IF NOT UseEnableWire THEN
	IF checkInitMultiplex() THEN
		RETURN;
	END_IF
ELSE
	IF NOT enableInstanceSet THEN
		RETURN;
	END_IF
END_IF
CASE _iState OF

RUN_DEVICE:
	//check if time are over
	IF TimeToRead < TICKS.GetTick(xDummy:= TRUE) AND haveToRead THEN 
		readRequest.request := TRUE;
		haveToRead := FALSE;
		TimeToReadOver := TRUE;
	END_IF
	IF UseEnableWire THEN
		IF NOT TimeToReadOver THEN
			RETURN;
		END_IF
	ELSE
		IF NOT checkReadTimeMultiplex(ADR(readRequest)) OR NOT TimeToReadOver THEN
			RETURN;
		END_IF
	END_IF
	ReadTime := TICKS.GetTick(xDummy:= TRUE);
	TimeToReadOver := FALSE;
	waitForDone := FALSE;
	IF NOT (setWire() = SET_SLAVE_NUM_RETURN.NUM_IO) AND UseEnableWire  THEN
		RETURN;
	END_IF
	//time over and on the bus... now read
	//read RH
	IF checkRead(pbyBuffer:= ADR(buffer), nBufferLen:= 3(*SIZEOF(buffer)*)) = ERROR_RET_VAL THEN
		ReadHuminityErrorRate := ReadHuminityErrorRate + 1;
		RETURN; 
	END_IF
	buffercrc[1] := buffer[0];
	buffercrc[2] := buffer[1];
	buffercrc[3] := buffer[2];
	buffercrc[0] := 0;
	crc := OSCAT_BASIC.CRC_GEN(
	PT:= ADR(buffercrc), 
	SIZE:= TO_INT(SIZEOF(buffercrc)), 
	PL:= 8, 
	PN:= 16#31, 
	INIT:= 0, 
	REV_IN:= FALSE, 
	REV_OUT:= FALSE, 
	XOR_OUT:= 0);
	IF crc = 0 THEN
		//checkRead(pbyBuffer:= ADR(buffer), nBufferLen:= SIZEOF(buffer));
		myData.Humidity := (((DWORD_TO_LREAL(OSCAT_BASIC.DWORD_OF_BYTE(B3:= 0, B2:= 0, B1:= buffer[0], B0:= buffer[1]))*125)/65536))-6;
		//read temp with command
		buffer[0] := COMMAND_READ_TEMP_FROM_PREVIOUS_RH;
		IF checkWrite(pbyBuffer:= ADR(buffer), nBufferLen:= 1) = ERROR_RET_VAL THEN //write just one command
			WriteTempReadErrorRate := WriteTempReadErrorRate + 1;
			RETURN; 
		END_IF
		IF checkRead(pbyBuffer:= ADR(buffer), nBufferLen:=2 (* SIZEOF(buffer)*)) = ERROR_RET_VAL THEN 
			ReadTempErrorRate := ReadTempErrorRate + 1;
		RETURN;
		END_IF
		myData.Temperatur := ((DWORD_TO_LREAL(OSCAT_BASIC.DWORD_OF_BYTE(B3:= 0, B2:= 0, B1:= buffer[0], B0:= buffer[1]))*175.72)/65536)-46.85;
		
		myData.absHumidity  := OSCAT_BUILDING.DEW_CON(RH:=LREAL_TO_REAL(myData.Humidity) , T:=LREAL_TO_REAL(myData.Temperatur) );
		myData.dewPoint := OSCAT_BUILDING.DEW_TEMP(RH:= LREAL_TO_REAL(myData.Humidity), T:=LREAL_TO_REAL(myData.Temperatur ));
	ELSE
		CRCErrorRate := CRCErrorRate + 1;
		goError(ReadWrite:=FALSE);
	END_IF
	releaseWire();

END_CASE
END_METHOD

METHOD BeforeWriteOutputs : INT
VAR

buffer:ARRAY[0..1]OF BYTE;

SystemTime: CAA.TICK;

END_VAR
SUPER^.BeforeWriteOutputs();

IF NOT UseEnableWire THEN
	IF checkInitMultiplex() THEN
		RETURN;
	END_IF
ELSE
	IF NOT enableInstanceSet THEN
		RETURN;
	END_IF
END_IF

CASE _iState OF
START_DEVICE:
	//check if time is over
	//writeRequest.request := requestOnInit;
	waitForDone := FALSE;
	writeRequest.request := TRUE;
	IF checkWriteTimeMultiplex(ADR(writeRequest)) = FALSE AND NOT UseEnableWire THEN
		RETURN;// i am not on the bus
	END_IF
	buffer[0] := COMMAND_WRITE_RESISTER_1;
	buffer[1] := controlRegister; 
	
	IF NOT (setWire() = SET_SLAVE_NUM_RETURN.NUM_IO) AND UseEnableWire THEN
		RETURN;
	END_IF
	checkWrite(pbyBuffer:= ADR(buffer), nBufferLen:= SIZEOF(buffer));
	IF _iState<>ERROR_DEVICE THEN
		_iState := RUN_DEVICE;
		//requestOnInit := FALSE;//init successful	
	END_IF
	releaseWire();		
RUN_DEVICE:
	SystemTime := TICKS.GetTick(xDummy:= TRUE);
	IF NextMeasuerment < SystemTime AND NOT waitForDone THEN 
		NextMeasuerment := timeMeasurment + SystemTime;
		waitForDone := TRUE; 
		writeRequest.request := TRUE;
		WriteRequestHuminity := TRUE;
	END_IF
	IF UseEnableWire THEN
		IF NOT WriteRequestHuminity THEN
			RETURN;
		END_IF
	ELSE
		IF NOT checkReadTimeMultiplex(ADR(writeRequest)) OR NOT WriteRequestHuminity THEN
			RETURN;
		END_IF
	END_IF
	WriteRequestHuminity := FALSE;
	//new time for Read the conversation
	TimeToRead := timePreset + TICKS.GetTick(xDummy:= TRUE);
	haveToRead := TRUE;

	IF NOT (setWire() = SET_SLAVE_NUM_RETURN.NUM_IO) AND UseEnableWire THEN
		RETURN;
	END_IF
	
	buffer[0] := COMMAND_MEASURE_RH_NO_HOLD_MASTER;
	IF checkWrite(pbyBuffer:= ADR(buffer), nBufferLen:= 1) = ERROR_RET_VAL THEN //write just one byte!
		WriteTempReadErrorRate := WriteTempReadErrorRate + 1;
	END_IF
	WriteTime := TICKS.GetTick(xDummy:= TRUE);
	releaseWire();
END_CASE
END_METHOD

METHOD Initialize : UDINT
VAR_INPUT
	wModuleType : UINT;
	dwInstance : UDINT;
	pConnector : POINTER TO IoConfigConnector;
END_VAR
VAR
	pParam: POINTER TO IoConfigParameter;		
	udiResult: UDINT;
	config:USINT;
END_VAR
SUPER^.Initialize(wModuleType, dwInstance, pConnector);
usiAddress := 16#40;
//get config
pParam := ConfigGetParameter(_pConnector, 20);



config:= IoStandard.ConfigGetParameterValueByte(pParam, ADR(udiResult));
CASE config OF//see Datasheet Page 26 for config
	//control Register --> resoulution
	0:	controlRegister := 2#1;
		timePreset := 8;//ms
	1:	controlRegister := 2#10000000;
		timePreset := 12;//ms
	2:	controlRegister := 2#10000001;
		timePreset := 12;//ms
	3:	controlRegister := 2#0;
		timePreset := 25;//ms
END_CASE

//time between Measurments
pParam := ConfigGetParameter(_pConnector, 21);
timeMeasurment := IoStandard.ConfigGetParameterValueDWord(pParam, ADR(udiResult));
//disable auto read
readRequest.timePreset := 16#FFFFFFFF; 
 
stateAfterError := START_DEVICE;
stateAfterInit := START_DEVICE;
END_METHOD

END_FUNCTION_BLOCK

// Function Blocks/BMP280
FUNCTION_BLOCK BMP280 EXTENDS I2C_BASE
VAR_INPUT

END_VAR
VAR_OUTPUT
	myData:BMP280Data;
	configWrong: BOOL;
END_VAR
VAR


	dig_T1: LREAL;
    dig_T2: LREAL;
    dig_T3: LREAL;
	 
    dig_P1: LREAL;
    dig_P2: LREAL;
    dig_P3: LREAL;
    dig_P4: LREAL;
    dig_P5: LREAL;
    dig_P6: LREAL;
    dig_P7: LREAL;
    dig_P8: LREAL;
    dig_P9: LREAL;

	t_fine:DINT;
	
	tempOversampling: USINT;
	pressureOversampling: USINT;

	iirFilter:USINT;
	standbyTime:USINT;
	controlRegister:BYTE;
	writeControlRegister:BOOL;
	operationMode:BYTE;
	//diffrenz for read the next value in ms
	nextForcedDiff:UDINT;
	//next time to write forced
	nextForced: CAA.TICK;
	//wrong device!
	wrongDevice: BOOL;


END_VAR
VAR_TEMP	
END_VAR

VAR CONSTANT 
	
BMP280_REGISTER_DIG_T1:USINT := 16#88;
BMP280_REGISTER_DIG_T2:USINT := 16#8A;
BMP280_REGISTER_DIG_T3:USINT := 16#8C;

BMP280_REGISTER_DIG_P1:USINT := 16#8E;
BMP280_REGISTER_DIG_P2:USINT := 16#90;
BMP280_REGISTER_DIG_P3:USINT := 16#92;
BMP280_REGISTER_DIG_P4:USINT := 16#94;
BMP280_REGISTER_DIG_P5:USINT := 16#96;
BMP280_REGISTER_DIG_P6:USINT := 16#98;
BMP280_REGISTER_DIG_P7:USINT := 16#9A;
BMP280_REGISTER_DIG_P8:USINT := 16#9C;
BMP280_REGISTER_DIG_P9:USINT := 16#9E;



BMP280_REGISTER_CHIPID:USINT := 16#D0;
BMP280_REGISTER_VERSION :USINT := 16#D1;
BMP280_REGISTER_SOFTRESET :USINT := 16#E0;


BMP280_REGISTER_CONTROL :USINT := 16#F4;
BMP280_REGISTER_CONFIG :USINT := 16#F5;
BMP280_REGISTER_PRESSURE_DATA :USINT := 16#F7;
BMP280_REGISTER_TEMP_DATA :USINT := 16#FA;

BMP_280_DEVICE_ID:USINT:=16#58;

TEMP_OVERSAMPLING_MAX:USINT:=5;
PRESSURE_OVERSAMPLING_MAX:USINT:=5;

IIR_FILTER_MAX:USINT:=4;
STANDBY_TIME_MAX:USINT:=7;
BMP280_NORMAL_MODE:USINT:=2#11;
BMP280_FORCED_MODE:USINT:=2#01;
BMP280_SLEEP_MODE:USINT:=2#00;

TEMPERATURE_OFF:UDINT:=16#80000;
PRESSURE_OFF:UDINT:=16#80000;




END_VAR

SUPER^();

CASE _iState OF
	RUN_DEVICE:
		IF operationMode = BMP280_FORCED_MODE THEN
			IF nextForced < TICKS.GetTick(xDummy:= TRUE) THEN
				//set next read
				nextForced := nextForcedDiff + TICKS.GetTick(xDummy:= TRUE);
				setForcedMode();
				
			END_IF 
		ELSE
			nextForced := nextForcedDiff + TICKS.GetTick(xDummy:= TRUE);
		END_IF
END_CASE

METHOD AfterReadInputs : INT
VAR
	sensorData: ARRAY[0..7] OF BYTE;	
	rawTempSensor:UDINT;
	rawTemp:LREAL;
	rawPressureSensor:UDINT;
	rawPressure:LREAL;
	rawHumiditySensor:UDINT;
	rawHumidity:LREAL;
	var1, var2, p, var_H:LREAL;
	tError, hError, pError: BOOL;
	//dd:LREAL;
END_VAR
SUPER^.AfterReadInputs();

IF checkInitMultiplex() THEN
	RETURN;
END_IF
CASE _iState OF
START_INIT:
	readRequest.request := TRUE;
	
	//check if time are over
	IF NOT checkReadTimeMultiplex(ADR(readRequest)) THEN
		RETURN;
	END_IF
	initCalibration();

	IF _iState<>ERROR_DEVICE THEN
		_iState := START_DEVICE;

	END_IF
RUN_DEVICE:
	//check if time are over
	IF NOT checkReadTimeMultiplex(ADR(readRequest)) THEN
		RETURN;
	END_IF
	(*read all sensor Data*)
	IF checkReadRegister(BMP280_REGISTER_PRESSURE_DATA, ADR(sensorData),6) < 0 THEN
		RETURN;
	END_IF
	
	rawTempSensor:=0;
	rawTempSensor:=SHL(BYTE_TO_UDINT(sensorData[3]),16);
	rawTempSensor:=rawTempSensor OR SHL(BYTE_TO_UDINT(sensorData[4]),8);
	rawTempSensor:=rawTempSensor OR BYTE_TO_UDINT(sensorData[5]);
	rawTempSensor:= SHR(rawTempSensor,4);
	//if Sensor value off and sensor switched on(no power)
	IF rawTempSensor = TEMPERATURE_OFF AND tempOversampling >0 THEN
		goError(ReadWrite := TRUE);
		RETURN;
	END_IF
	IF rawTempSensor <> 16#80000 THEN
		rawTemp:=UDINT_TO_REAL(rawTempSensor);
		var1  := (rawTemp/16384.0 - dig_T1/1024.0) * dig_T2;
		var2  := ((rawTemp/131072.0 - dig_T1/8192.0) *   (rawTemp/131072.0 -  dig_T1/8192.0)) * dig_T3;
		t_fine := LREAL_TO_DINT(var1 + var2);
		myData.Temperatur  := (var1 + var2) / 5120.0;
		
	ELSE
		myData.Temperatur:=0.0;
		
	END_IF
	//Calculate pressure
	rawPressureSensor:=0;
	rawPressureSensor:=SHL(BYTE_TO_UDINT(sensorData[0]),16);
	rawPressureSensor:=rawPressureSensor OR SHL(BYTE_TO_UDINT(sensorData[1]),8);
	rawPressureSensor:=rawPressureSensor OR BYTE_TO_UDINT(sensorData[2]);
	rawPressureSensor:= SHR(rawPressureSensor,4);
	IF rawPressureSensor = PRESSURE_OFF AND pressureOversampling >0 THEN
		goError(ReadWrite := TRUE);
		RETURN;
	END_IF
	IF rawPressureSensor <> 16#80000 THEN
		rawPressure:=UDINT_TO_REAL(rawPressureSensor);
		var1 := (DINT_TO_LREAL(t_fine)/2.0) - 64000.0;
		var2 := var1 * var1 * (dig_P6) / 32768.0;
		var2 := var2 + var1 * (dig_P5) * 2.0;
		var2 := (var2/4.0)+((dig_P4) * 65536.0);
		var1 := ((dig_P3) * var1 * var1 / 524288.0 + (dig_P2) * var1) / 524288.0;
		var1 := (1.0 + var1 / 32768.0)*(dig_P1);
		IF var1 = 0.0 THEN
			myData.Pressure := 0.0;
		ELSE	
			p := 1048576.0 - rawPressure;
			p := (p - (var2 / 4096.0)) * 6250.0 / var1;
			var1 := (dig_P9) * p * p / 2147483648.0;
			var2 := p * (dig_P8) / 32768.0;
			p := p + (var1 + var2 + (dig_P7)) / 16.0;
			myData.Pressure := p; 	
		END_IF
  	ELSE
		myData.Pressure :=0.0;
	END_IF

	
END_CASE
END_METHOD

METHOD Initialize : UDINT
VAR_INPUT
	wModuleType : UINT;
	dwInstance : UDINT;
	pConnector : POINTER TO IoConfigConnector;
END_VAR
VAR
	pParam: POINTER TO IoConfigParameter;		
	udiResult: UDINT;
	byte1:byte;
END_VAR
SUPER^.Initialize(wModuleType, dwInstance, pConnector);

IF usiAddress = 0 THEN
	usiAddress := 16#77;
END_IF


pParam := ConfigGetParameter(_pConnector, 20);
tempOversampling:= IoStandard.ConfigGetParameterValueByte(pParam, ADR(udiResult));
IF tempOversampling > TEMP_OVERSAMPLING_MAX THEN
	 tempOversampling := TEMP_OVERSAMPLING_MAX;
	configWrong := TRUE; 
END_IF
pParam := ConfigGetParameter(_pConnector, 21);
pressureOversampling:= IoStandard.ConfigGetParameterValueByte(pParam, ADR(udiResult));
IF pressureOversampling > PRESSURE_OVERSAMPLING_MAX THEN
	pressureOversampling := PRESSURE_OVERSAMPLING_MAX;
	configWrong := TRUE;
END_IF

pParam := ConfigGetParameter(_pConnector, 22);
iirFilter:= IoStandard.ConfigGetParameterValueByte(pParam, ADR(udiResult));
IF iirFilter > IIR_FILTER_MAX THEN
	iirFilter := IIR_FILTER_MAX;
	configWrong := TRUE;
END_IF
pParam := ConfigGetParameter(_pConnector, 23);
standbyTime:= IoStandard.ConfigGetParameterValueByte(pParam, ADR(udiResult));
IF standbyTime > STANDBY_TIME_MAX THEN
	standbyTime := STANDBY_TIME_MAX;
	configWrong := TRUE;
END_IF

pParam := ConfigGetParameter(_pConnector, 24);
nextForcedDiff:= IoStandard.ConfigGetParameterValueDWord(pParam, ADR(udiResult));
IF nextForcedDiff = 0  THEN
	operationMode := BMP280_NORMAL_MODE;
ELSE
	operationMode := BMP280_FORCED_MODE;
END_IF


errorFromChild := configWrong;

stateAfterError := START_INIT;
stateAfterInit := START_INIT;
END_METHOD

METHOD BeforeWriteOutputs : INT
VAR

END_VAR
SUPER^.BeforeWriteOutputs();

IF checkInitMultiplex() THEN
	RETURN;
END_IF

CASE _iState OF
START_DEVICE:
	//check if time is over
	//writeRequest.request := requestOnInit;
	writeRequest.request := TRUE;
	IF checkWriteTimeMultiplex(ADR(writeRequest)) = FALSE  THEN
		RETURN;// i am not on the bus
	END_IF
	
	initDevice();
	IF _iState<>ERROR_DEVICE THEN
		_iState := RUN_DEVICE;
		//requestOnInit := FALSE;//init successful	
	END_IF
	
RUN_DEVICE:
	IF checkWriteTimeMultiplex(ADR(writeRequest)) = FALSE  THEN
		RETURN;// i am not on the bus
	END_IF
	IF writeControlRegister THEN
		IF checkWrite8(BMP280_REGISTER_CONTROL,controlRegister) < 0 THEN
			RETURN;
		ELSE
			writeControlRegister := FALSE;
			IF operationMode = BMP280_FORCED_MODE THEN
				readRequest.request := TRUE;
			END_IF
		END_IF
	END_IF
	
	
END_CASE
END_METHOD

METHOD initCalibration
VAR_INPUT
END_VAR
VAR
	byte1: BYTE;
	byte2: BYTE;
	x: INT;
	tint:INT;
	tuint:UINT;
	tusint:USINT;
	tsint:SINT;
	
END_VAR
(*read calibration values from BMP 280 *)
//check device
IF checkReadRegister(BMP280_REGISTER_CHIPID, ADR(tusint),1) < 0 THEN
	RETURN;
END_IF
IF tusint <> BMP_280_DEVICE_ID THEN//wrong device --> go error
	goError(ReadWrite:= TRUE);
	wrongDevice := TRUE;
	RETURN;
ELSE
	wrongDevice := FALSE;
END_IF
IF checkReadRegister(BMP280_REGISTER_DIG_T1, ADR(tuint),2) < 0 THEN
	RETURN;
END_IF
dig_T1 := UINT_TO_LREAL(tuint);
IF checkReadRegister(BMP280_REGISTER_DIG_T2, ADR(tint),2) < 0 THEN
	RETURN;
END_IF 
dig_T2 := INT_TO_LREAL(tint);
IF checkReadRegister(BMP280_REGISTER_DIG_T3, ADR(tint),2) < 0 THEN
	RETURN;
END_IF
dig_T3 := INT_TO_LREAL(tint);

IF checkReadRegister(BMP280_REGISTER_DIG_P1, ADR(tuint),2) <0 THEN
	RETURN;
END_IF
dig_P1 := UINT_TO_LREAL(tuint);
IF checkReadRegister(BMP280_REGISTER_DIG_P2, ADR(tint),2) < 0 THEN
	RETURN;
END_IF
dig_P2 := INT_TO_LREAL(tint);
IF checkReadRegister(BMP280_REGISTER_DIG_P3, ADR(tint),2) < 0 THEN
	RETURN;
END_IF
dig_P3 := INT_TO_LREAL(tint);
IF checkReadRegister(BMP280_REGISTER_DIG_P4, ADR(tint),2) < 0 THEN
	RETURN;
END_IF
dig_P4 := INT_TO_LREAL(tint);
IF checkReadRegister(BMP280_REGISTER_DIG_P5, ADR(tint),2) < 0 THEN
	RETURN;
END_IF
dig_P5 := INT_TO_LREAL(tint);
IF checkReadRegister(BMP280_REGISTER_DIG_P6, ADR(tint),2) < 0 THEN
	RETURN;
END_IF
dig_P6 := INT_TO_LREAL(tint);
IF checkReadRegister(BMP280_REGISTER_DIG_P7, ADR(tint),2) < 0 THEN
	RETURN;
END_IF
dig_P7 := INT_TO_LREAL(tint);
IF checkReadRegister(BMP280_REGISTER_DIG_P8, ADR(tint),2) < 0 THEN
	RETURN;
END_IF
dig_P8 := INT_TO_LREAL(tint);
IF checkReadRegister(BMP280_REGISTER_DIG_P9, ADR(tint),2) < 0 THEN
	RETURN;
END_IF
dig_P9 := INT_TO_LREAL(tint);
END_METHOD

METHOD initDevice : INT
VAR_INPUT
END_VAR
IF checkWrite8(BMP280_REGISTER_CONFIG, (SHL(standbyTime,5)OR SHL(iirFilter,2))) < 0 THEN
	RETURN;		
END_IF
	

calcControlRegister();
IF checkWrite8(BMP280_REGISTER_CONTROL,controlRegister) < 0 THEN
	RETURN;
END_IF
END_METHOD

METHOD setForcedMode
VAR_INPUT
END_VAR
operationMode := BMP280_FORCED_MODE;
calcControlRegister();
writeControlRegister := TRUE;
writeRequest.request := TRUE;
END_METHOD

METHOD calcControlRegister
VAR_INPUT
END_VAR
controlRegister := SHL(tempOversampling,5)OR SHL(pressureOversampling,2)OR operationMode;
END_METHOD

END_FUNCTION_BLOCK

// VISU/SSD1306
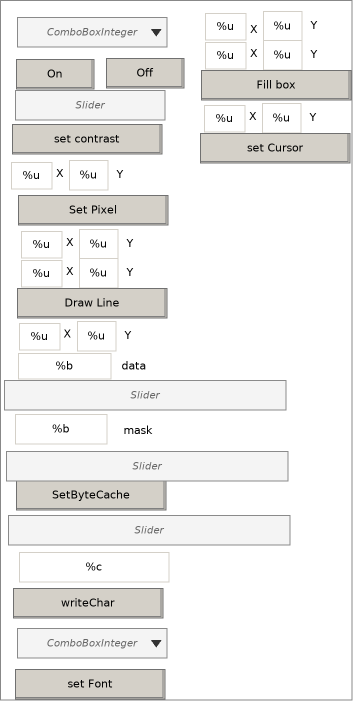
VISUALIZATION SSD1306  // 353x701
VAR_IN_OUT
	LCD:SSD1306;
END_VAR
VAR
	contrast:BYTE;
	x:USINT;
	y:USINT;
	x1Line:USINT;
	y1Line:USINT;
	x2Line:USINT;
	y2Line:USINT;
	xSetByte:USINT;
	ySetByte:USINT;
	dataSetByte:BYTE;
	maskSetByte:BYTE;
	mode:LCD_MODES:=1;
	c:BYTE:=16#41;
	aktFont:SOFT_FONT_NUMS;
	x1Box:USINT;
	x2Box:USINT;
	y1Box:USINT;
	y2Box:USINT;
	xCursor:USINT;
	yCursor:USINT;
END_VAR
    Button (16,59 78x30), "On"
        OnMouseClick: execute { LCD.DisplayOn(); }
    Button (106,58 78x30), "Off"
        OnMouseClick: execute { LCD.DisplayOff(); }
    Slider (15,90 150x30), variable: contrast, scale 0..255
    Button (12,124 150x30), "set contrast"
        OnMouseClick: execute { LCD.SetContrast(contrast:= contrast); }
    Textfield (11,162 41x27), "%u", text variable: x, input disabled if: false
        OnMouseClick: write the text variable via Default, min 0, max 127, format %u
    Label (49,159 22x29), "X"
    Textfield (69,160 39x30), "%u", text variable: y, input disabled if: false
        OnMouseClick: write the text variable via Default, min 0, max 63, format %u
    Label (109,160 22x29), "Y"
    Button (18,195 150x30), "Set Pixel"
        OnMouseClick: execute { LCD.SetPixelCache(xPos:= x, yPos:= y, mode:= mode); LCD.WriteCacheToLcd(); }
    Textfield (21,231 41x27), "%u", text variable: x1Line, input disabled if: false
        OnMouseClick: write the text variable via Default, min 0, max 127, format %u
    Label (59,228 22x29), "X"
    Textfield (79,229 39x30), "%u", text variable: y1Line, input disabled if: false
        OnMouseClick: write the text variable via Default, min 0, max 63, format %u
    Label (119,229 22x29), "Y"
    Textfield (21,260 41x27), "%u", text variable: x2Line, input disabled if: false
        OnMouseClick: write the text variable via Default, min 0, max 127, format %u
    Label (59,257 22x29), "X"
    Textfield (79,258 39x30), "%u", text variable: y2Line, input disabled if: false
        OnMouseClick: write the text variable via Default, min 0, max 63, format %u
    Label (119,258 22x29), "Y"
    Button (17,288 150x30), "Draw Line"
        OnMouseClick: execute {
            LCD.DrawLine(
            	x1:= x1Line,
            	y1:= y1Line,
            	x2:=x2Line ,
            	y2:= y2Line,
            	mode:= mode);
            LCD.WriteCacheToLcd();
        }
    Textfield (19,323 41x27), "%u", text variable: xSetByte, input disabled if: false
        OnMouseClick: write the text variable via Default, min 0, max 127, format %u
    Label (57,320 21x28), "X"
    Textfield (77,321 39x30), "%u", text variable: ySetByte, input disabled if: false
        OnMouseClick: write the text variable via Default, min 0, max 63, format %u
    Label (117,321 22x29), "Y"
    Textfield (18,353 93x26), "%b", text variable: dataSetByte, input disabled if: false
        OnMouseClick: write the text variable via Default, min 0, max 255, format %b
    Textfield (15,414 92x30), "%b", text variable: MaskSetByte, input disabled if: false
        OnMouseClick: write the text variable via Default, min 0, max 255, format %b
    Label (116,352 36x28), "data"
    Label (115,416 46x29), "mask"
    Button (16,480 150x30), "SetByteCache"
        OnMouseClick: execute {
            LCD.SetByteCache(
            	xpos:= xSetByte,
            	ypos:= ySetByte,
            	data:= dataSetByte,
            	mask:= maskSetByte,
            	mode:= mode);
            LCD.WriteCacheToLcd();
        }
    ComboBoxInteger (17,17 150x30), variable: mode
    Button (13,588 150x30), "writeChar"
        OnMouseClick: execute { LCD.WriteChar(c:= c, mode:= mode); LCD.WriteCacheToLcd(); }
    Slider (8,515 282x30), variable: c, scale 0..255
    Textfield (19,552 150x30), "%c", text variable: c
    ComboBoxInteger (17,628 150x30), variable: aktFont, text list: 'SOFT_FONT_NAMES'
    Button (15,669 150x30), "set Font"
        OnMouseClick: execute { LCD.SetSoftFont(aktFont); }
    Textfield (205,13 41x27), "%u", text variable: x1Box, input disabled if: false
        OnMouseClick: write the text variable via Default, min 0, max 127, format %u
    Textfield (263,11 39x30), "%u", text variable: y1Box, input disabled if: false
        OnMouseClick: write the text variable via Default, min 0, max 63, format %u
    Label (303,11 22x29), "Y"
    Textfield (205,42 41x27), "%u", text variable: x2Box, input disabled if: false
        OnMouseClick: write the text variable via Default, min 0, max 127, format %u
    Label (243,39 22x29), "X"
    Textfield (263,40 39x30), "%u", text variable: y2Box, input disabled if: false
        OnMouseClick: write the text variable via Default, min 0, max 63, format %u
    Label (303,40 22x29), "Y"
    Button (201,70 150x30), "Fill box"
        OnMouseClick: execute {
            LCD.FillBox(
            	x1:= x1Box,
            	y1:= y1Box,
            	x2:= x2Box,
            	y2:= y2Box,
            	mode:= mode);
            LCD.WriteCacheToLcd();
        }
    Textfield (204,105 41x27), "%u", text variable: xCursor, input disabled if: false
        OnMouseClick: write the text variable via Default, min 0, max 127, format %u
    Label (242,102 22x29), "X"
    Textfield (262,103 39x30), "%u", text variable: yCursor, input disabled if: false
        OnMouseClick: write the text variable via Default, min 0, max 63, format %u
    Label (302,103 22x29), "Y"
    Button (200,133 150x30), "set Cursor"
        OnMouseClick: execute { LCD.SetCursor(x:= xCursor, y:= yCursor); }
    Label (243,15 22x29), "X"
    Slider (4,380 282x30), variable: dataSetByte, scale 0..255
    Slider (6,451 282x30), variable: MaskSetByte, scale 0..255
END_VISUALIZATION

(* text list SOFT_FONT_NAMES (id | default)
  0 | 4X6
  1 | 5X8
  2 | 5X12
  3 | 6X8
  4 | 6X10
  5 | 7X12
  6 | 7X12B
  7 | 8X8
  8 | 8X12
  9 | 8X14
  10 | 10X16
  11 | 12X16
  12 | 16X8
  13 | 16X12
  14 | 16X26
   |  *)
